# B&R Automation Studio project MotionTestBenchMaster (part 54)

```iecst
                               VAR_DOS_SEQ.Device.LTJ203.ALR_HighLimitEn := FALSE;                                     (* STEP: 89 Hema Tank Level*)
                               VAR_DOS_SEQ.Device.LTJ203.ALR_HighLimitSP := 0;
                               VAR_DOS_SEQ.Device.LTJ203.ALR_LowLimitEn := FALSE;
                               VAR_DOS_SEQ.Device.LTJ203.ALR_LowLimitSP := 0;
                               VAR_DOS_SEQ.Device.LTJ203.SP := 0;
                               VAR_DOS_SEQ.Device.LTJ203.CMP := 0;
                               VAR_DOS_SEQ.Device.LTJ203.MinDev := 0;
                               VAR_DOS_SEQ.Device.LTJ203.MaxDev := 0;

                               VAR_DOS_SEQ.Device.TTJ203.ALR_HighLimitEn := FALSE;                                     (* STEP: 89 Hema Tank Temperature*)
                               VAR_DOS_SEQ.Device.TTJ203.ALR_HighLimitSP := 0;
                               VAR_DOS_SEQ.Device.TTJ203.ALR_LowLimitEn := FALSE;
                               VAR_DOS_SEQ.Device.TTJ203.ALR_LowLimitSP := 0;
                               VAR_DOS_SEQ.Device.TTJ203.SP := 0;
                               VAR_DOS_SEQ.Device.TTJ203.CMP := 0;
                               VAR_DOS_SEQ.Device.TTJ203.MinDev := 0;
                               VAR_DOS_SEQ.Device.TTJ203.MaxDev := 0;

                               VAR_DOS_SEQ.Device.LSJ200.ALR := FALSE;                                                 (* STEP: 89 *)
                               VAR_DOS_SEQ.Device.LSJ200.WAIT_OFF := FALSE;
                               VAR_DOS_SEQ.Device.LSJ200.WAIT_ON := FALSE;

                               VAR_DOS_SEQ.Device.LSJ201.ALR := FALSE;                                                 (* STEP: 89 *)
                               VAR_DOS_SEQ.Device.LSJ201.WAIT_OFF := FALSE;
                               VAR_DOS_SEQ.Device.LSJ201.WAIT_ON := FALSE;

                               VAR_DOS_SEQ.Device.LSJ202.ALR := FALSE;                                                 (* STEP: 89 *)
                               VAR_DOS_SEQ.Device.LSJ202.WAIT_OFF := FALSE;
                               VAR_DOS_SEQ.Device.LSJ202.WAIT_ON := FALSE;

                               VAR_DOS_SEQ.Device.FSJ201.ALR := FALSE;                                                 (* STEP: 89 *)
                               VAR_DOS_SEQ.Device.FSJ201.WAIT_OFF := FALSE;
                               VAR_DOS_SEQ.Device.FSJ201.WAIT_ON := FALSE;

                               VAR_DOS_SEQ.Device.FSJ202.ALR := FALSE;                                                 (* STEP: 89 *)
                               VAR_DOS_SEQ.Device.FSJ202.WAIT_OFF := FALSE;
                               VAR_DOS_SEQ.Device.FSJ202.WAIT_ON := FALSE;

                               VAR_DOS_SEQ.Mem.PBAbortEnable := FALSE;                                                 (* STEP: 89 PB Abort Sequence Enable*)
                               VAR_DOS_SEQ.Mem.PBStopEnable := FALSE;                                                  (* STEP: 89 PB Stop Sequence Enable*)
                               VAR_DOS_SEQ.Mem.PBStartEnable := FALSE;                                                 (* STEP: 89 PB Start Sequence Enable*)
                               VAR_DOS_SEQ.Mem.ContainersStop := TRUE;                                                 (* STEP: 89 *)
                               VAR_DOS_SEQ.Mem.MachineStart := FALSE;                                                  (* STEP: 89 *)
                               VAR_DOS_SEQ.Mem.MachineStop := TRUE;                                                    (* STEP: 89 *)
                               VAR_DOS_SEQ.Mem.DummyBottles := FALSE;                                                  (* STEP: 89 Dummy Bottle Install*)
                               VAR_DOS_SEQ.Mem.PositioningRequest := TRUE;                                             (* STEP: 89 Request of Cam Positioning at height SP of Sequncer*)
                               VAR_DOS_SEQ.Mem.COP_Cycle := TRUE;                                                      (* STEP: 89 COP Cycle Check Requested*)
                               VAR_DOS_SEQ.Mem.LapsCounter := FALSE;                                                   (* STEP: 89 *)
                               VAR_DOS_SEQ.Mem.ValveOpening := FALSE;                                                  (* STEP: 89 *)
                               VAR_DOS_SEQ.Mem.CopAfterCipRequest := FALSE;                                            (* STEP: 89 Request Of Cop After Cip*)

                               VAR_DOS_SEQ.ITC.CIP_CleaningRequest := FALSE;                                           (* STEP: 89 To CIP -> Request of Solution Sending*)
                               VAR_DOS_SEQ.ITC.CIP_Alarm := FALSE;                                                     (* STEP: 89 To CIP -> Critical Alarm Present*)
                               VAR_DOS_SEQ.ITC.CIP_RinseEnded := FALSE;                                                (* STEP: 89 To CIP -> Rinse Finished*)
                               VAR_DOS_SEQ.ITC.CIP_ChangeEnded := FALSE;                                               (* STEP: 89 To CIP -> Change Finished*)
                               VAR_DOS_SEQ.ITC.CIP_DrainRunning := FALSE;                                              (* STEP: 89 To CIP -> Drain Cycle Running*)
                               VAR_DOS_SEQ.ITC.CIP_RinseRunning := FALSE;                                              (* STEP: 89 To CIP -> Rinse Cycle Running*)
                               VAR_DOS_SEQ.ITC.CIP_CleaningRunning := FALSE;                                           (* STEP: 89 To CIP -> Cleaning Cycle Running*)
                               VAR_DOS_SEQ.ITC.CIP_DrainEnded := FALSE;                                                (* STEP: 89 To CIP -> Drain Finished*)
                               VAR_DOS_SEQ.ITC.CIP_FloodingEnded := FALSE;                                             (* STEP: 89 To CIP -> Flooding Finished*)
                               VAR_DOS_SEQ.ITC.CIP_FlipEnable := FALSE;                                                (* STEP: 89 *)
                               VAR_DOS_SEQ.ITC.CIP_CycleEnded := FALSE;                                                (* STEP: 89 *)

                               VAR_DOS_SEQ.ITC.PROD_ReadyForHeating := FALSE;                                          (* STEP: 89 To PASTO -> Filler Ready for Production (Heating)*)
                               VAR_DOS_SEQ.ITC.PROD_DoserInTemperature := FALSE;                                       (* STEP: 89 To PASTO -> Filler Temperature OK (After Heating)*)
                               VAR_DOS_SEQ.ITC.PROD_ProductRequest := FALSE;                                           (* STEP: 89 To PASTO -> Product Request*)
                               VAR_DOS_SEQ.ITC.PROD_DoserOnFillingMode := FALSE;                                       (* STEP: 89 To PASTO -> Product Consumend -Filling Valve Opening*)
                               VAR_DOS_SEQ.ITC.PROD_EndProductionCompleted := FALSE;                                   (* STEP: 89 To PASTO -> End Production Done*)
                               VAR_DOS_SEQ.ITC.PROD_ProductRecoveryEnd := FALSE;                                       (* STEP: 89 To PASTO -> Product Recovery End*)
                               VAR_DOS_SEQ.ITC.PROD_WaterRequestAfterProd := FALSE;                                    (* STEP: 89 To PASTO -> Water Request For Filler Rinse Afetr Production*)

                       90: (* COP in Execution *)

                               VAR_DOS_SEQ.Device.PPJ201_PID.PID_Enable := FALSE;                                      (* STEP: 90 Doser Recovery Pump*)
                               VAR_DOS_SEQ.Device.PPJ201_PID.PID_Mode := FALSE;
                               VAR_DOS_SEQ.Device.PPJ201_PID.Auto_SP_Value := 0;
                               VAR_DOS_SEQ.Device.PPJ201_PID.FIX_Value := 0;

                               VAR_DOS_SEQ.Device.PPJ202_PID.PID_Enable := FALSE;                                      (* STEP: 90 Doser Recovery Pump*)
                               VAR_DOS_SEQ.Device.PPJ202_PID.PID_Mode := FALSE;
                               VAR_DOS_SEQ.Device.PPJ202_PID.Auto_SP_Value := 0;
                               VAR_DOS_SEQ.Device.PPJ202_PID.FIX_Value := 0;

                               VAR_DOS_SEQ.Device.PPJ203_PID.PID_Enable := FALSE;                                      (* STEP: 90 Diaphragm Pump for Recovery pulp*)
                               VAR_DOS_SEQ.Device.PPJ203_PID.PID_Mode := FALSE;
                               VAR_DOS_SEQ.Device.PPJ203_PID.Auto_SP_Value := 0;
                               VAR_DOS_SEQ.Device.PPJ203_PID.FIX_Value := 0;

                               VAR_DOS_SEQ.Device.MMJ201_PID.PID_Enable := FALSE;                                      (* STEP: 90 Shaker Motor*)
                               VAR_DOS_SEQ.Device.MMJ201_PID.PID_Mode := FALSE;
                               VAR_DOS_SEQ.Device.MMJ201_PID.Auto_SP_Value := 0;
                               VAR_DOS_SEQ.Device.MMJ201_PID.FIX_Value := 0;

                               VAR_DOS_SEQ.Device.RVJ201_PID.PID_Enable := FALSE;                                      (* STEP: 90 *)
                               VAR_DOS_SEQ.Device.RVJ201_PID.PID_Mode := FALSE;
                               VAR_DOS_SEQ.Device.RVJ201_PID.Auto_SP_Value := 0;
                               VAR_DOS_SEQ.Device.RVJ201_PID.FIX_Value := 0;

                               VAR_DOS_SEQ.Device.AVJ201.AutoCnd := FALSE;                                             (* STEP: 90 Inlet Valve*)
                               VAR_DOS_SEQ.Device.AVJ201.EnableCnd := FALSE;
                               VAR_DOS_SEQ.Device.AVJ210.AutoCnd := FALSE;                                             (* STEP: 90 Washing Duct Valve*)
                               VAR_DOS_SEQ.Device.AVJ210.EnableCnd := FALSE;
                               VAR_DOS_SEQ.Device.AVJ211.AutoCnd := FALSE;                                             (* STEP: 90 Sprayball Valve*)
                               VAR_DOS_SEQ.Device.AVJ211.EnableCnd := FALSE;
                               VAR_DOS_SEQ.Device.AVJ212.AutoCnd := FALSE;                                             (* STEP: 90 *)
                               VAR_DOS_SEQ.Device.AVJ212.EnableCnd := FALSE;
                               VAR_DOS_SEQ.Device.AVJ215.AutoCnd := TRUE;                                              (* STEP: 90 Atmospheric drain valve*)
                               VAR_DOS_SEQ.Device.AVJ215.EnableCnd := FALSE;
                               VAR_DOS_SEQ.Device.AVJ216.AutoCnd := FALSE;                                             (* STEP: 90 Recirculation Valve*)
                               VAR_DOS_SEQ.Device.AVJ216.EnableCnd := FALSE;
                               VAR_DOS_SEQ.Device.AVJ217.AutoCnd := TRUE;                                              (* STEP: 90 Tank Hema Drain Valve*)
                               VAR_DOS_SEQ.Device.AVJ217.EnableCnd := FALSE;
                               VAR_DOS_SEQ.Device.AVJ218.AutoCnd := FALSE;                                             (* STEP: 90 Recirculation Valve*)
                               VAR_DOS_SEQ.Device.AVJ218.EnableCnd := FALSE;
                               VAR_DOS_SEQ.Device.AVJ221.AutoCnd := FALSE;                                             (* STEP: 90 Inlet Loop Valve*)
                               VAR_DOS_SEQ.Device.AVJ221.EnableCnd := FALSE;
                               VAR_DOS_SEQ.Device.AVJ230.AutoCnd := FALSE;                                             (* STEP: 90 *)
                               VAR_DOS_SEQ.Device.AVJ230.EnableCnd := FALSE;
                               VAR_DOS_SEQ.Device.AVJ231.AutoCnd := FALSE;                                             (* STEP: 90 *)
                               VAR_DOS_SEQ.Device.AVJ231.EnableCnd := FALSE;
                               VAR_DOS_SEQ.Device.AVJ232.AutoCnd := FALSE;                                             (* STEP: 90 *)
                               VAR_DOS_SEQ.Device.AVJ232.EnableCnd := FALSE;
                               VAR_DOS_SEQ.Device.AVJ233.AutoCnd := FALSE;                                             (* STEP: 90 *)
                               VAR_DOS_SEQ.Device.AVJ233.EnableCnd := FALSE;
                               VAR_DOS_SEQ.Device.AVJ234.AutoCnd := FALSE;                                             (* STEP: 90 *)
                               VAR_DOS_SEQ.Device.AVJ234.EnableCnd := FALSE;
                               VAR_DOS_SEQ.Device.AVJ235.AutoCnd := FALSE;                                             (* STEP: 90 *)
                               VAR_DOS_SEQ.Device.AVJ235.EnableCnd := FALSE;

                               VAR_DOS_SEQ.Device.LTJ203.ALR_HighLimitEn := FALSE;                                     (* STEP: 90 Hema Tank Level*)
                               VAR_DOS_SEQ.Device.LTJ203.ALR_HighLimitSP := 0;
                               VAR_DOS_SEQ.Device.LTJ203.ALR_LowLimitEn := FALSE;
                               VAR_DOS_SEQ.Device.LTJ203.ALR_LowLimitSP := 0;
                               VAR_DOS_SEQ.Device.LTJ203.SP := 0;
                               VAR_DOS_SEQ.Device.LTJ203.CMP := 0;
                               VAR_DOS_SEQ.Device.LTJ203.MinDev := 0;
                               VAR_DOS_SEQ.Device.LTJ203.MaxDev := 0;

                               VAR_DOS_SEQ.Device.TTJ203.ALR_HighLimitEn := FALSE;                                     (* STEP: 90 Hema Tank Temperature*)
                               VAR_DOS_SEQ.Device.TTJ203.ALR_HighLimitSP := 0;
                               VAR_DOS_SEQ.Device.TTJ203.ALR_LowLimitEn := FALSE;
                               VAR_DOS_SEQ.Device.TTJ203.ALR_LowLimitSP := 0;
                               VAR_DOS_SEQ.Device.TTJ203.SP := 0;
                               VAR_DOS_SEQ.Device.TTJ203.CMP := 0;
                               VAR_DOS_SEQ.Device.TTJ203.MinDev := 0;
                               VAR_DOS_SEQ.Device.TTJ203.MaxDev := 0;

                               VAR_DOS_SEQ.Device.LSJ200.ALR := FALSE;                                                 (* STEP: 90 *)
                               VAR_DOS_SEQ.Device.LSJ200.WAIT_OFF := FALSE;
                               VAR_DOS_SEQ.Device.LSJ200.WAIT_ON := FALSE;

                               VAR_DOS_SEQ.Device.LSJ201.ALR := FALSE;                                                 (* STEP: 90 *)
                               VAR_DOS_SEQ.Device.LSJ201.WAIT_OFF := FALSE;
                               VAR_DOS_SEQ.Device.LSJ201.WAIT_ON := FALSE;

                               VAR_DOS_SEQ.Device.LSJ202.ALR := FALSE;                                                 (* STEP: 90 *)
                               VAR_DOS_SEQ.Device.LSJ202.WAIT_OFF := FALSE;
                               VAR_DOS_SEQ.Device.LSJ202.WAIT_ON := FALSE;

                               VAR_DOS_SEQ.Device.FSJ201.ALR := FALSE;                                                 (* STEP: 90 *)
                               VAR_DOS_SEQ.Device.FSJ201.WAIT_OFF := FALSE;
                               VAR_DOS_SEQ.Device.FSJ201.WAIT_ON := FALSE;

                               VAR_DOS_SEQ.Device.FSJ202.ALR := FALSE;                                                 (* STEP: 90 *)
                               VAR_DOS_SEQ.Device.FSJ202.WAIT_OFF := FALSE;
                               VAR_DOS_SEQ.Device.FSJ202.WAIT_ON := FALSE;

                               VAR_DOS_SEQ.Mem.PBAbortEnable := FALSE;                                                 (* STEP: 90 PB Abort Sequence Enable*)
                               VAR_DOS_SEQ.Mem.PBStopEnable := FALSE;                                                  (* STEP: 90 PB Stop Sequence Enable*)
                               VAR_DOS_SEQ.Mem.PBStartEnable := FALSE;                                                 (* STEP: 90 PB Start Sequence Enable*)
                               VAR_DOS_SEQ.Mem.ContainersStop := TRUE;                                                 (* STEP: 90 *)
                               VAR_DOS_SEQ.Mem.MachineStart := TRUE;                                                   (* STEP: 90 *)
                               VAR_DOS_SEQ.Mem.MachineStop := FALSE;                                                   (* STEP: 90 *)
                               VAR_DOS_SEQ.Mem.DummyBottles := FALSE;                                                  (* STEP: 90 Dummy Bottle Install*)
                               VAR_DOS_SEQ.Mem.PositioningRequest := FALSE;                                            (* STEP: 90 Request of Cam Positioning at height SP of Sequncer*)
                               VAR_DOS_SEQ.Mem.COP_Cycle := TRUE;                                                      (* STEP: 90 COP Cycle Check Requested*)
                               VAR_DOS_SEQ.Mem.LapsCounter := FALSE;                                                   (* STEP: 90 *)
                               VAR_DOS_SEQ.Mem.ValveOpening := FALSE;                                                  (* STEP: 90 *)
                               VAR_DOS_SEQ.Mem.CopAfterCipRequest := FALSE;                                            (* STEP: 90 Request Of Cop After Cip*)

                               VAR_DOS_SEQ.ITC.CIP_CleaningRequest := FALSE;                                           (* STEP: 90 To CIP -> Request of Solution Sending*)
                               VAR_DOS_SEQ.ITC.CIP_Alarm := FALSE;                                                     (* STEP: 90 To CIP -> Critical Alarm Present*)
                               VAR_DOS_SEQ.ITC.CIP_RinseEnded := FALSE;                                                (* STEP: 90 To CIP -> Rinse Finished*)
                               VAR_DOS_SEQ.ITC.CIP_ChangeEnded := FALSE;                                               (* STEP: 90 To CIP -> Change Finished*)
                               VAR_DOS_SEQ.ITC.CIP_DrainRunning := FALSE;                                              (* STEP: 90 To CIP -> Drain Cycle Running*)
                               VAR_DOS_SEQ.ITC.CIP_RinseRunning := FALSE;                                              (* STEP: 90 To CIP -> Rinse Cycle Running*)
                               VAR_DOS_SEQ.ITC.CIP_CleaningRunning := FALSE;                                           (* STEP: 90 To CIP -> Cleaning Cycle Running*)
                               VAR_DOS_SEQ.ITC.CIP_DrainEnded := FALSE;                                                (* STEP: 90 To CIP -> Drain Finished*)
                               VAR_DOS_SEQ.ITC.CIP_FloodingEnded := FALSE;                                             (* STEP: 90 To CIP -> Flooding Finished*)
                               VAR_DOS_SEQ.ITC.CIP_FlipEnable := FALSE;                                                (* STEP: 90 *)
                               VAR_DOS_SEQ.ITC.CIP_CycleEnded := FALSE;                                                (* STEP: 90 *)

                               VAR_DOS_SEQ.ITC.PROD_ReadyForHeating := FALSE;                                          (* STEP: 90 To PASTO -> Filler Ready for Production (Heating)*)
                               VAR_DOS_SEQ.ITC.PROD_DoserInTemperature := FALSE;                                       (* STEP: 90 To PASTO -> Filler Temperature OK (After Heating)*)
                               VAR_DOS_SEQ.ITC.PROD_ProductRequest := FALSE;                                           (* STEP: 90 To PASTO -> Product Request*)
                               VAR_DOS_SEQ.ITC.PROD_DoserOnFillingMode := FALSE;                                       (* STEP: 90 To PASTO -> Product Consumend -Filling Valve Opening*)
                               VAR_DOS_SEQ.ITC.PROD_EndProductionCompleted := FALSE;                                   (* STEP: 90 To PASTO -> End Production Done*)
                               VAR_DOS_SEQ.ITC.PROD_ProductRecoveryEnd := FALSE;                                       (* STEP: 90 To PASTO -> Product Recovery End*)
                               VAR_DOS_SEQ.ITC.PROD_WaterRequestAfterProd := FALSE;                                    (* STEP: 90 To PASTO -> Water Request For Filler Rinse Afetr Production*)
//change
                       91: (* Drain Recovery Skid *)

								VAR_DOS_SEQ.Device.PPJ201_PID.PID_Enable := FALSE;                                      (* STEP: 91 Doser Recovery Pump*)
								VAR_DOS_SEQ.Device.PPJ201_PID.PID_Mode := FALSE;
								VAR_DOS_SEQ.Device.PPJ201_PID.Auto_SP_Value := 0;
								VAR_DOS_SEQ.Device.PPJ201_PID.FIX_Value := 0;

								VAR_DOS_SEQ.Device.PPJ202_PID.PID_Enable := FALSE;                                      (* STEP: 91 Doser Recovery Pump*)
								VAR_DOS_SEQ.Device.PPJ202_PID.PID_Mode := FALSE;
								VAR_DOS_SEQ.Device.PPJ202_PID.Auto_SP_Value := 0;
								VAR_DOS_SEQ.Device.PPJ202_PID.FIX_Value := 0;

								VAR_DOS_SEQ.Device.PPJ203_PID.PID_Enable := FALSE;                                      (* STEP: 91 Diaphragm Pump for Recovery pulp*)
								VAR_DOS_SEQ.Device.PPJ203_PID.PID_Mode := FALSE;
								VAR_DOS_SEQ.Device.PPJ203_PID.Auto_SP_Value := 0;
								VAR_DOS_SEQ.Device.PPJ203_PID.FIX_Value := 0;

								VAR_DOS_SEQ.Device.MMJ201_PID.PID_Enable := FALSE;                                      (* STEP: 91 Shaker Motor*)
								VAR_DOS_SEQ.Device.MMJ201_PID.PID_Mode := FALSE;
								VAR_DOS_SEQ.Device.MMJ201_PID.Auto_SP_Value := 0;
								VAR_DOS_SEQ.Device.MMJ201_PID.FIX_Value := 0;

								VAR_DOS_SEQ.Device.RVJ201_PID.PID_Enable := FALSE;                                      (* STEP: 91 *)
								VAR_DOS_SEQ.Device.RVJ201_PID.PID_Mode := FALSE;
								VAR_DOS_SEQ.Device.RVJ201_PID.Auto_SP_Value := 0;
								VAR_DOS_SEQ.Device.RVJ201_PID.FIX_Value := 0;

								VAR_DOS_SEQ.Device.AVJ201.AutoCnd := FALSE;                                             (* STEP: 91 Inlet Valve*)
								VAR_DOS_SEQ.Device.AVJ201.EnableCnd := FALSE;
								VAR_DOS_SEQ.Device.AVJ210.AutoCnd := FALSE;                                             (* STEP: 91 Washing Duct Valve*)
								VAR_DOS_SEQ.Device.AVJ210.EnableCnd := FALSE;
								VAR_DOS_SEQ.Device.AVJ211.AutoCnd := FALSE;                                             (* STEP: 91 Sprayball Valve*)
								VAR_DOS_SEQ.Device.AVJ211.EnableCnd := FALSE;
								VAR_DOS_SEQ.Device.AVJ212.AutoCnd := FALSE;                                             (* STEP: 91 *)
								VAR_DOS_SEQ.Device.AVJ212.EnableCnd := FALSE;
								VAR_DOS_SEQ.Device.AVJ215.AutoCnd := TRUE;                                              (* STEP: 91 Atmospheric drain valve*)
								VAR_DOS_SEQ.Device.AVJ215.EnableCnd := FALSE;
								VAR_DOS_SEQ.Device.AVJ216.AutoCnd := FALSE;                                             (* STEP: 91 Recirculation Valve*)
								VAR_DOS_SEQ.Device.AVJ216.EnableCnd := FALSE;
								VAR_DOS_SEQ.Device.AVJ217.AutoCnd := TRUE;                                              (* STEP: 91 Tank Hema Drain Valve*)
								VAR_DOS_SEQ.Device.AVJ217.EnableCnd := FALSE;
								VAR_DOS_SEQ.Device.AVJ218.AutoCnd := FALSE;                                             (* STEP: 91 Recirculation Valve*)
								VAR_DOS_SEQ.Device.AVJ218.EnableCnd := FALSE;
								VAR_DOS_SEQ.Device.AVJ221.AutoCnd := FALSE;                                             (* STEP: 91 Inlet Loop Valve*)
								VAR_DOS_SEQ.Device.AVJ221.EnableCnd := FALSE;
								VAR_DOS_SEQ.Device.AVJ230.AutoCnd := FALSE;                                             (* STEP: 91 *)
								VAR_DOS_SEQ.Device.AVJ230.EnableCnd := FALSE;
								VAR_DOS_SEQ.Device.AVJ231.AutoCnd := FALSE;                                             (* STEP: 91 *)
								VAR_DOS_SEQ.Device.AVJ231.EnableCnd := FALSE;
								VAR_DOS_SEQ.Device.AVJ232.AutoCnd := TRUE;                                             (* STEP: 91 *)
								VAR_DOS_SEQ.Device.AVJ232.EnableCnd := FALSE;
								VAR_DOS_SEQ.Device.AVJ233.AutoCnd := FALSE;                                             (* STEP: 91 *)
								VAR_DOS_SEQ.Device.AVJ233.EnableCnd := FALSE;
								VAR_DOS_SEQ.Device.AVJ234.AutoCnd := FALSE;                                             (* STEP: 91 *)
								VAR_DOS_SEQ.Device.AVJ234.EnableCnd := FALSE;
								VAR_DOS_SEQ.Device.AVJ235.AutoCnd := TRUE;                                             (* STEP: 91 *)
								VAR_DOS_SEQ.Device.AVJ235.EnableCnd := FALSE;

								VAR_DOS_SEQ.Device.LTJ203.ALR_HighLimitEn := FALSE;                                     (* STEP: 91 Hema Tank Level*)
								VAR_DOS_SEQ.Device.LTJ203.ALR_HighLimitSP := 0;
								VAR_DOS_SEQ.Device.LTJ203.ALR_LowLimitEn := FALSE;
								VAR_DOS_SEQ.Device.LTJ203.ALR_LowLimitSP := 0;
								VAR_DOS_SEQ.Device.LTJ203.SP := 0;
								VAR_DOS_SEQ.Device.LTJ203.CMP := 0;
								VAR_DOS_SEQ.Device.LTJ203.MinDev := 0;
								VAR_DOS_SEQ.Device.LTJ203.MaxDev := 0;

								VAR_DOS_SEQ.Device.TTJ203.ALR_HighLimitEn := FALSE;                                     (* STEP: 91 Hema Tank Temperature*)
								VAR_DOS_SEQ.Device.TTJ203.ALR_HighLimitSP := 0;
								VAR_DOS_SEQ.Device.TTJ203.ALR_LowLimitEn := FALSE;
								VAR_DOS_SEQ.Device.TTJ203.ALR_LowLimitSP := 0;
								VAR_DOS_SEQ.Device.TTJ203.SP := 0;
								VAR_DOS_SEQ.Device.TTJ203.CMP := 0;
								VAR_DOS_SEQ.Device.TTJ203.MinDev := 0;
								VAR_DOS_SEQ.Device.TTJ203.MaxDev := 0;

								VAR_DOS_SEQ.Device.LSJ200.ALR := FALSE;                                                 (* STEP: 91 *)
								VAR_DOS_SEQ.Device.LSJ200.WAIT_OFF := FALSE;
								VAR_DOS_SEQ.Device.LSJ200.WAIT_ON := FALSE;

								VAR_DOS_SEQ.Device.LSJ201.ALR := FALSE;                                                 (* STEP: 91 *)
								VAR_DOS_SEQ.Device.LSJ201.WAIT_OFF := FALSE;
								VAR_DOS_SEQ.Device.LSJ201.WAIT_ON := FALSE;

								VAR_DOS_SEQ.Device.LSJ202.ALR := FALSE;                                                 (* STEP: 91 *)
								VAR_DOS_SEQ.Device.LSJ202.WAIT_OFF := FALSE;
								VAR_DOS_SEQ.Device.LSJ202.WAIT_ON := FALSE;

								VAR_DOS_SEQ.Device.FSJ201.ALR := FALSE;                                                 (* STEP: 91 *)
								VAR_DOS_SEQ.Device.FSJ201.WAIT_OFF := FALSE;
								VAR_DOS_SEQ.Device.FSJ201.WAIT_ON := FALSE;

								VAR_DOS_SEQ.Device.FSJ202.ALR := FALSE;                                                 (* STEP: 91 *)
								VAR_DOS_SEQ.Device.FSJ202.WAIT_OFF := FALSE;
								VAR_DOS_SEQ.Device.FSJ202.WAIT_ON := FALSE;

								VAR_DOS_SEQ.Mem.PBAbortEnable := FALSE;                                                 (* STEP: 91 PB Abort Sequence Enable*)
								VAR_DOS_SEQ.Mem.PBStopEnable := FALSE;                                                  (* STEP: 91 PB Stop Sequence Enable*)
								VAR_DOS_SEQ.Mem.PBStartEnable := FALSE;                                                 (* STEP: 91 PB Start Sequence Enable*)
								VAR_DOS_SEQ.Mem.ContainersStop := TRUE;                                                 (* STEP: 91 *)
								VAR_DOS_SEQ.Mem.MachineStart := FALSE;                                                   (* STEP: 91 *)
								VAR_DOS_SEQ.Mem.MachineStop := TRUE;                                                   (* STEP: 91 *)
								VAR_DOS_SEQ.Mem.DummyBottles := FALSE;                                                  (* STEP: 91 Dummy Bottle Install*)
								VAR_DOS_SEQ.Mem.PositioningRequest := FALSE;                                            (* STEP: 91 Request of Cam Positioning at height SP of Sequncer*)
								VAR_DOS_SEQ.Mem.COP_Cycle := TRUE;                                                      (* STEP: 91 COP Cycle Check Requested*)
								VAR_DOS_SEQ.Mem.LapsCounter := FALSE;                                                   (* STEP: 91 *)
								VAR_DOS_SEQ.Mem.ValveOpening := FALSE;                                                  (* STEP: 91 *)
								VAR_DOS_SEQ.Mem.CopAfterCipRequest := FALSE;                                            (* STEP: 91 Request Of Cop After Cip*)

								VAR_DOS_SEQ.ITC.CIP_CleaningRequest := FALSE;                                           (* STEP: 91 To CIP -> Request of Solution Sending*)
								VAR_DOS_SEQ.ITC.CIP_Alarm := FALSE;                                                     (* STEP: 91 To CIP -> Critical Alarm Present*)
								VAR_DOS_SEQ.ITC.CIP_RinseEnded := FALSE;                                                (* STEP: 91 To CIP -> Rinse Finished*)
								VAR_DOS_SEQ.ITC.CIP_ChangeEnded := FALSE;                                               (* STEP: 91 To CIP -> Change Finished*)
								VAR_DOS_SEQ.ITC.CIP_DrainRunning := FALSE;                                              (* STEP: 91 To CIP -> Drain Cycle Running*)
								VAR_DOS_SEQ.ITC.CIP_RinseRunning := FALSE;                                              (* STEP: 91 To CIP -> Rinse Cycle Running*)
								VAR_DOS_SEQ.ITC.CIP_CleaningRunning := FALSE;                                           (* STEP: 91 To CIP -> Cleaning Cycle Running*)
								VAR_DOS_SEQ.ITC.CIP_DrainEnded := FALSE;                                                (* STEP: 91 To CIP -> Drain Finished*)
								VAR_DOS_SEQ.ITC.CIP_FloodingEnded := FALSE;                                             (* STEP: 91 To CIP -> Flooding Finished*)
								VAR_DOS_SEQ.ITC.CIP_FlipEnable := FALSE;                                                (* STEP: 91 *)
								VAR_DOS_SEQ.ITC.CIP_CycleEnded := FALSE;                                                (* STEP: 91 *)

								VAR_DOS_SEQ.ITC.PROD_ReadyForHeating := FALSE;                                          (* STEP: 91 To PASTO -> Filler Ready for Production (Heating)*)
								VAR_DOS_SEQ.ITC.PROD_DoserInTemperature := FALSE;                                       (* STEP: 91 To PASTO -> Filler Temperature OK (After Heating)*)
								VAR_DOS_SEQ.ITC.PROD_ProductRequest := FALSE;                                           (* STEP: 91 To PASTO -> Product Request*)
								VAR_DOS_SEQ.ITC.PROD_DoserOnFillingMode := FALSE;                                       (* STEP: 91 To PASTO -> Product Consumend -Filling Valve Opening*)
								VAR_DOS_SEQ.ITC.PROD_EndProductionCompleted := FALSE;                                   (* STEP: 91 To PASTO -> End Production Done*)
								VAR_DOS_SEQ.ITC.PROD_ProductRecoveryEnd := FALSE;                                       (* STEP: 91 To PASTO -> Product Recovery End*)
								VAR_DOS_SEQ.ITC.PROD_WaterRequestAfterProd := FALSE;                                    (* STEP: 91 To PASTO -> Water Request For Filler Rinse Afetr Production*)

                       92: (* CIP -Wait Dummy Bottles Disinsertion *)

                               VAR_DOS_SEQ.Device.PPJ201_PID.PID_Enable := FALSE;                                      (* STEP: 92 Doser Recovery Pump*)
                               VAR_DOS_SEQ.Device.PPJ201_PID.PID_Mode := FALSE;
                               VAR_DOS_SEQ.Device.PPJ201_PID.Auto_SP_Value := 0;
                               VAR_DOS_SEQ.Device.PPJ201_PID.FIX_Value := 0;

                               VAR_DOS_SEQ.Device.PPJ202_PID.PID_Enable := FALSE;                                      (* STEP: 92 Doser Recovery Pump*)
                               VAR_DOS_SEQ.Device.PPJ202_PID.PID_Mode := FALSE;
                               VAR_DOS_SEQ.Device.PPJ202_PID.Auto_SP_Value := 0;
                               VAR_DOS_SEQ.Device.PPJ202_PID.FIX_Value := 0;

                               VAR_DOS_SEQ.Device.PPJ203_PID.PID_Enable := FALSE;                                      (* STEP: 92 Diaphragm Pump for Recovery pulp*)
                               VAR_DOS_SEQ.Device.PPJ203_PID.PID_Mode := FALSE;
                               VAR_DOS_SEQ.Device.PPJ203_PID.Auto_SP_Value := 0;
                               VAR_DOS_SEQ.Device.PPJ203_PID.FIX_Value := 0;

                               VAR_DOS_SEQ.Device.MMJ201_PID.PID_Enable := FALSE;                                      (* STEP: 92 Shaker Motor*)
                               VAR_DOS_SEQ.Device.MMJ201_PID.PID_Mode := FALSE;
                               VAR_DOS_SEQ.Device.MMJ201_PID.Auto_SP_Value := 0;
                               VAR_DOS_SEQ.Device.MMJ201_PID.FIX_Value := 0;

                               VAR_DOS_SEQ.Device.RVJ201_PID.PID_Enable := FALSE;                                      (* STEP: 92 *)
                               VAR_DOS_SEQ.Device.RVJ201_PID.PID_Mode := FALSE;
                               VAR_DOS_SEQ.Device.RVJ201_PID.Auto_SP_Value := 0;
                               VAR_DOS_SEQ.Device.RVJ201_PID.FIX_Value := 0;

                               VAR_DOS_SEQ.Device.AVJ201.AutoCnd := FALSE;                                             (* STEP: 92 Inlet Valve*)
                               VAR_DOS_SEQ.Device.AVJ201.EnableCnd := FALSE;
                               VAR_DOS_SEQ.Device.AVJ210.AutoCnd := FALSE;                                             (* STEP: 92 Washing Duct Valve*)
                               VAR_DOS_SEQ.Device.AVJ210.EnableCnd := FALSE;
                               VAR_DOS_SEQ.Device.AVJ211.AutoCnd := FALSE;                                             (* STEP: 92 Sprayball Valve*)
                               VAR_DOS_SEQ.Device.AVJ211.EnableCnd := FALSE;
                               VAR_DOS_SEQ.Device.AVJ212.AutoCnd := FALSE;                                             (* STEP: 92 *)
                               VAR_DOS_SEQ.Device.AVJ212.EnableCnd := FALSE;
                               VAR_DOS_SEQ.Device.AVJ215.AutoCnd := FALSE;                                             (* STEP: 92 Atmospheric drain valve*)
                               VAR_DOS_SEQ.Device.AVJ215.EnableCnd := FALSE;
                               VAR_DOS_SEQ.Device.AVJ216.AutoCnd := FALSE;                                             (* STEP: 92 Recirculation Valve*)
                               VAR_DOS_SEQ.Device.AVJ216.EnableCnd := FALSE;
                               VAR_DOS_SEQ.Device.AVJ217.AutoCnd := FALSE;                                             (* STEP: 92 Tank Hema Drain Valve*)
                               VAR_DOS_SEQ.Device.AVJ217.EnableCnd := FALSE;
                               VAR_DOS_SEQ.Device.AVJ218.AutoCnd := FALSE;                                             (* STEP: 92 Recirculation Valve*)
                               VAR_DOS_SEQ.Device.AVJ218.EnableCnd := FALSE;
                               VAR_DOS_SEQ.Device.AVJ221.AutoCnd := FALSE;                                             (* STEP: 92 Inlet Loop Valve*)
                               VAR_DOS_SEQ.Device.AVJ221.EnableCnd := FALSE;
                               VAR_DOS_SEQ.Device.AVJ230.AutoCnd := FALSE;                                             (* STEP: 92 *)
                               VAR_DOS_SEQ.Device.AVJ230.EnableCnd := FALSE;
                               VAR_DOS_SEQ.Device.AVJ231.AutoCnd := FALSE;                                             (* STEP: 92 *)
                               VAR_DOS_SEQ.Device.AVJ231.EnableCnd := FALSE;
                               VAR_DOS_SEQ.Device.AVJ232.AutoCnd := FALSE;                                             (* STEP: 92 *)
                               VAR_DOS_SEQ.Device.AVJ232.EnableCnd := FALSE;
                               VAR_DOS_SEQ.Device.AVJ233.AutoCnd := FALSE;                                             (* STEP: 92 *)
                               VAR_DOS_SEQ.Device.AVJ233.EnableCnd := FALSE;
                               VAR_DOS_SEQ.Device.AVJ234.AutoCnd := FALSE;                                             (* STEP: 92 *)
                               VAR_DOS_SEQ.Device.AVJ234.EnableCnd := FALSE;
                               VAR_DOS_SEQ.Device.AVJ235.AutoCnd := FALSE;                                             (* STEP: 92 *)
                               VAR_DOS_SEQ.Device.AVJ235.EnableCnd := FALSE;

                               VAR_DOS_SEQ.Device.LTJ203.ALR_HighLimitEn := FALSE;                                     (* STEP: 92 Hema Tank Level*)
                               VAR_DOS_SEQ.Device.LTJ203.ALR_HighLimitSP := 0;
                               VAR_DOS_SEQ.Device.LTJ203.ALR_LowLimitEn := FALSE;
                               VAR_DOS_SEQ.Device.LTJ203.ALR_LowLimitSP := 0;
                               VAR_DOS_SEQ.Device.LTJ203.SP := 0;
                               VAR_DOS_SEQ.Device.LTJ203.CMP := 0;
                               VAR_DOS_SEQ.Device.LTJ203.MinDev := 0;
                               VAR_DOS_SEQ.Device.LTJ203.MaxDev := 0;

                               VAR_DOS_SEQ.Device.TTJ203.ALR_HighLimitEn := FALSE;                                     (* STEP: 92 Hema Tank Temperature*)
                               VAR_DOS_SEQ.Device.TTJ203.ALR_HighLimitSP := 0;
                               VAR_DOS_SEQ.Device.TTJ203.ALR_LowLimitEn := FALSE;
                               VAR_DOS_SEQ.Device.TTJ203.ALR_LowLimitSP := 0;
                               VAR_DOS_SEQ.Device.TTJ203.SP := 0;
                               VAR_DOS_SEQ.Device.TTJ203.CMP := 0;
                               VAR_DOS_SEQ.Device.TTJ203.MinDev := 0;
                               VAR_DOS_SEQ.Device.TTJ203.MaxDev := 0;

                               VAR_DOS_SEQ.Device.LSJ200.ALR := FALSE;                                                 (* STEP: 92 *)
                               VAR_DOS_SEQ.Device.LSJ200.WAIT_OFF := FALSE;
                               VAR_DOS_SEQ.Device.LSJ200.WAIT_ON := FALSE;

                               VAR_DOS_SEQ.Device.LSJ201.ALR := FALSE;                                                 (* STEP: 92 *)
                               VAR_DOS_SEQ.Device.LSJ201.WAIT_OFF := FALSE;
                               VAR_DOS_SEQ.Device.LSJ201.WAIT_ON := FALSE;

                               VAR_DOS_SEQ.Device.LSJ202.ALR := FALSE;                                                 (* STEP: 92 *)
                               VAR_DOS_SEQ.Device.LSJ202.WAIT_OFF := FALSE;
                               VAR_DOS_SEQ.Device.LSJ202.WAIT_ON := FALSE;

                               VAR_DOS_SEQ.Device.FSJ201.ALR := FALSE;                                                 (* STEP: 92 *)
                               VAR_DOS_SEQ.Device.FSJ201.WAIT_OFF := FALSE;
                               VAR_DOS_SEQ.Device.FSJ201.WAIT_ON := FALSE;

                               VAR_DOS_SEQ.Device.FSJ202.ALR := FALSE;                                                 (* STEP: 92 *)
                               VAR_DOS_SEQ.Device.FSJ202.WAIT_OFF := FALSE;
                               VAR_DOS_SEQ.Device.FSJ202.WAIT_ON := FALSE;

                               VAR_DOS_SEQ.Mem.PBAbortEnable := FALSE;                                                 (* STEP: 92 PB Abort Sequence Enable*)
                               VAR_DOS_SEQ.Mem.PBStopEnable := FALSE;                                                  (* STEP: 92 PB Stop Sequence Enable*)
                               VAR_DOS_SEQ.Mem.PBStartEnable := FALSE;                                                 (* STEP: 92 PB Start Sequence Enable*)
                               VAR_DOS_SEQ.Mem.ContainersStop := FALSE;                                                (* STEP: 92 *)
                               VAR_DOS_SEQ.Mem.MachineStart := FALSE;                                                  (* STEP: 92 *)
                               VAR_DOS_SEQ.Mem.MachineStop := FALSE;                                                   (* STEP: 92 *)
                               VAR_DOS_SEQ.Mem.DummyBottles := FALSE;                                                  (* STEP: 92 Dummy Bottle Install*)
                               VAR_DOS_SEQ.Mem.PositioningRequest := FALSE;                                            (* STEP: 92 Request of Cam Positioning at height SP of Sequncer*)
                               VAR_DOS_SEQ.Mem.COP_Cycle := FALSE;                                                     (* STEP: 92 COP Cycle Check Requested*)
                               VAR_DOS_SEQ.Mem.LapsCounter := FALSE;                                                   (* STEP: 92 *)
                               VAR_DOS_SEQ.Mem.ValveOpening := FALSE;                                                  (* STEP: 92 *)
                               VAR_DOS_SEQ.Mem.CopAfterCipRequest := FALSE;                                            (* STEP: 92 Request Of Cop After Cip*)

                               VAR_DOS_SEQ.ITC.CIP_CleaningRequest := FALSE;                                           (* STEP: 92 To CIP -> Request of Solution Sending*)
                               VAR_DOS_SEQ.ITC.CIP_Alarm := FALSE;                                                     (* STEP: 92 To CIP -> Critical Alarm Present*)
                               VAR_DOS_SEQ.ITC.CIP_RinseEnded := FALSE;                                                (* STEP: 92 To CIP -> Rinse Finished*)
                               VAR_DOS_SEQ.ITC.CIP_ChangeEnded := FALSE;                                               (* STEP: 92 To CIP -> Change Finished*)
                               VAR_DOS_SEQ.ITC.CIP_DrainRunning := FALSE;                                              (* STEP: 92 To CIP -> Drain Cycle Running*)
                               VAR_DOS_SEQ.ITC.CIP_RinseRunning := FALSE;                                              (* STEP: 92 To CIP -> Rinse Cycle Running*)
                               VAR_DOS_SEQ.ITC.CIP_CleaningRunning := FALSE;                                           (* STEP: 92 To CIP -> Cleaning Cycle Running*)
                               VAR_DOS_SEQ.ITC.CIP_DrainEnded := FALSE;                                                (* STEP: 92 To CIP -> Drain Finished*)
                               VAR_DOS_SEQ.ITC.CIP_FloodingEnded := FALSE;                                             (* STEP: 92 To CIP -> Flooding Finished*)
                               VAR_DOS_SEQ.ITC.CIP_FlipEnable := FALSE;                                                (* STEP: 92 *)
                               VAR_DOS_SEQ.ITC.CIP_CycleEnded := FALSE;                                                (* STEP: 92 *)

                               VAR_DOS_SEQ.ITC.PROD_ReadyForHeating := FALSE;                                          (* STEP: 92 To PASTO -> Filler Ready for Production (Heating)*)
                               VAR_DOS_SEQ.ITC.PROD_DoserInTemperature := FALSE;                                       (* STEP: 92 To PASTO -> Filler Temperature OK (After Heating)*)
                               VAR_DOS_SEQ.ITC.PROD_ProductRequest := FALSE;                                           (* STEP: 92 To PASTO -> Product Request*)
                               VAR_DOS_SEQ.ITC.PROD_DoserOnFillingMode := FALSE;                                       (* STEP: 92 To PASTO -> Product Consumend -Filling Valve Opening*)
                               VAR_DOS_SEQ.ITC.PROD_EndProductionCompleted := FALSE;                                   (* STEP: 92 To PASTO -> End Production Done*)
                               VAR_DOS_SEQ.ITC.PROD_ProductRecoveryEnd := FALSE;                                       (* STEP: 92 To PASTO -> Product Recovery End*)
                               VAR_DOS_SEQ.ITC.PROD_WaterRequestAfterProd := FALSE;                                    (* STEP: 92 To PASTO -> Water Request For Filler Rinse Afetr Production*)

                       93..94: (* Spare Steps *)

                       95: (* CIP - Stopped *)

                               VAR_DOS_SEQ.Device.PPJ201_PID.PID_Enable := FALSE;                                      (* STEP: 95 Doser Recovery Pump*)
                               VAR_DOS_SEQ.Device.PPJ201_PID.PID_Mode := FALSE;
                               VAR_DOS_SEQ.Device.PPJ201_PID.Auto_SP_Value := 0;
                               VAR_DOS_SEQ.Device.PPJ201_PID.FIX_Value := 0;

                               VAR_DOS_SEQ.Device.PPJ202_PID.PID_Enable := FALSE;                                      (* STEP: 95 Doser Recovery Pump*)
                               VAR_DOS_SEQ.Device.PPJ202_PID.PID_Mode := FALSE;
                               VAR_DOS_SEQ.Device.PPJ202_PID.Auto_SP_Value := 0;
                               VAR_DOS_SEQ.Device.PPJ202_PID.FIX_Value := 0;

                               VAR_DOS_SEQ.Device.PPJ203_PID.PID_Enable := FALSE;                                      (* STEP: 95 Diaphragm Pump for Recovery pulp*)
                               VAR_DOS_SEQ.Device.PPJ203_PID.PID_Mode := FALSE;
                               VAR_DOS_SEQ.Device.PPJ203_PID.Auto_SP_Value := 0;
                               VAR_DOS_SEQ.Device.PPJ203_PID.FIX_Value := 0;

                               VAR_DOS_SEQ.Device.MMJ201_PID.PID_Enable := FALSE;                                      (* STEP: 95 Shaker Motor*)
                               VAR_DOS_SEQ.Device.MMJ201_PID.PID_Mode := FALSE;
                               VAR_DOS_SEQ.Device.MMJ201_PID.Auto_SP_Value := 0;
                               VAR_DOS_SEQ.Device.MMJ201_PID.FIX_Value := 0;

                               VAR_DOS_SEQ.Device.RVJ201_PID.PID_Enable := FALSE;                                      (* STEP: 95 *)
                               VAR_DOS_SEQ.Device.RVJ201_PID.PID_Mode := FALSE;
                               VAR_DOS_SEQ.Device.RVJ201_PID.Auto_SP_Value := 0;
                               VAR_DOS_SEQ.Device.RVJ201_PID.FIX_Value := 0;

                               VAR_DOS_SEQ.Device.AVJ201.AutoCnd := FALSE;                                             (* STEP: 95 Inlet Valve*)
                               VAR_DOS_SEQ.Device.AVJ201.EnableCnd := FALSE;
                               VAR_DOS_SEQ.Device.AVJ210.AutoCnd := FALSE;                                             (* STEP: 95 Washing Duct Valve*)
                               VAR_DOS_SEQ.Device.AVJ210.EnableCnd := FALSE;
                               VAR_DOS_SEQ.Device.AVJ211.AutoCnd := FALSE;                                             (* STEP: 95 Sprayball Valve*)
                               VAR_DOS_SEQ.Device.AVJ211.EnableCnd := FALSE;
                               VAR_DOS_SEQ.Device.AVJ212.AutoCnd := FALSE;                                             (* STEP: 95 *)
                               VAR_DOS_SEQ.Device.AVJ212.EnableCnd := FALSE;
                               VAR_DOS_SEQ.Device.AVJ215.AutoCnd := FALSE;                                             (* STEP: 95 Atmospheric drain valve*)
                               VAR_DOS_SEQ.Device.AVJ215.EnableCnd := FALSE;
                               VAR_DOS_SEQ.Device.AVJ216.AutoCnd := FALSE;                                             (* STEP: 95 Recirculation Valve*)
                               VAR_DOS_SEQ.Device.AVJ216.EnableCnd := FALSE;
                               VAR_DOS_SEQ.Device.AVJ217.AutoCnd := FALSE;                                             (* STEP: 95 Tank Hema Drain Valve*)
                               VAR_DOS_SEQ.Device.AVJ217.EnableCnd := FALSE;
                               VAR_DOS_SEQ.Device.AVJ218.AutoCnd := FALSE;                                             (* STEP: 95 Recirculation Valve*)
                               VAR_DOS_SEQ.Device.AVJ218.EnableCnd := FALSE;
                               VAR_DOS_SEQ.Device.AVJ221.AutoCnd := FALSE;                                             (* STEP: 95 Inlet Loop Valve*)
                               VAR_DOS_SEQ.Device.AVJ221.EnableCnd := FALSE;
                               VAR_DOS_SEQ.Device.AVJ230.AutoCnd := FALSE;                                             (* STEP: 95 *)
                               VAR_DOS_SEQ.Device.AVJ230.EnableCnd := FALSE;
                               VAR_DOS_SEQ.Device.AVJ231.AutoCnd := FALSE;                                             (* STEP: 95 *)
                               VAR_DOS_SEQ.Device.AVJ231.EnableCnd := FALSE;
                               VAR_DOS_SEQ.Device.AVJ232.AutoCnd := FALSE;                                             (* STEP: 95 *)
                               VAR_DOS_SEQ.Device.AVJ232.EnableCnd := FALSE;
                               VAR_DOS_SEQ.Device.AVJ233.AutoCnd := FALSE;                                             (* STEP: 95 *)
                               VAR_DOS_SEQ.Device.AVJ233.EnableCnd := FALSE;
                               VAR_DOS_SEQ.Device.AVJ234.AutoCnd := FALSE;                                             (* STEP: 95 *)
                               VAR_DOS_SEQ.Device.AVJ234.EnableCnd := FALSE;
                               VAR_DOS_SEQ.Device.AVJ235.AutoCnd := FALSE;                                             (* STEP: 95 *)
                               VAR_DOS_SEQ.Device.AVJ235.EnableCnd := FALSE;

                               VAR_DOS_SEQ.Device.LTJ203.ALR_HighLimitEn := FALSE;                                     (* STEP: 95 Hema Tank Level*)
                               VAR_DOS_SEQ.Device.LTJ203.ALR_HighLimitSP := 0;
                               VAR_DOS_SEQ.Device.LTJ203.ALR_LowLimitEn := FALSE;
                               VAR_DOS_SEQ.Device.LTJ203.ALR_LowLimitSP := 0;
                               VAR_DOS_SEQ.Device.LTJ203.SP := 0;
                               VAR_DOS_SEQ.Device.LTJ203.CMP := 0;
                               VAR_DOS_SEQ.Device.LTJ203.MinDev := 0;
                               VAR_DOS_SEQ.Device.LTJ203.MaxDev := 0;

                               VAR_DOS_SEQ.Device.TTJ203.ALR_HighLimitEn := FALSE;                                     (* STEP: 95 Hema Tank Temperature*)
                               VAR_DOS_SEQ.Device.TTJ203.ALR_HighLimitSP := 0;
                               VAR_DOS_SEQ.Device.TTJ203.ALR_LowLimitEn := FALSE;
                               VAR_DOS_SEQ.Device.TTJ203.ALR_LowLimitSP := 0;
                               VAR_DOS_SEQ.Device.TTJ203.SP := 0;
                               VAR_DOS_SEQ.Device.TTJ203.CMP := 0;
                               VAR_DOS_SEQ.Device.TTJ203.MinDev := 0;
                               VAR_DOS_SEQ.Device.TTJ203.MaxDev := 0;

                               VAR_DOS_SEQ.Device.LSJ200.ALR := FALSE;                                                 (* STEP: 95 *)
                               VAR_DOS_SEQ.Device.LSJ200.WAIT_OFF := FALSE;
                               VAR_DOS_SEQ.Device.LSJ200.WAIT_ON := FALSE;

                               VAR_DOS_SEQ.Device.LSJ201.ALR := FALSE;                                                 (* STEP: 95 *)
                               VAR_DOS_SEQ.Device.LSJ201.WAIT_OFF := FALSE;
                               VAR_DOS_SEQ.Device.LSJ201.WAIT_ON := FALSE;

                               VAR_DOS_SEQ.Device.LSJ202.ALR := FALSE;                                                 (* STEP: 95 *)
                               VAR_DOS_SEQ.Device.LSJ202.WAIT_OFF := FALSE;
                               VAR_DOS_SEQ.Device.LSJ202.WAIT_ON := FALSE;

                               VAR_DOS_SEQ.Device.FSJ201.ALR := FALSE;                                                 (* STEP: 95 *)
                               VAR_DOS_SEQ.Device.FSJ201.WAIT_OFF := FALSE;
                               VAR_DOS_SEQ.Device.FSJ201.WAIT_ON := FALSE;

                               VAR_DOS_SEQ.Device.FSJ202.ALR := FALSE;                                                 (* STEP: 95 *)
                               VAR_DOS_SEQ.Device.FSJ202.WAIT_OFF := FALSE;
                               VAR_DOS_SEQ.Device.FSJ202.WAIT_ON := FALSE;

                               VAR_DOS_SEQ.Mem.PBAbortEnable := TRUE;                                                  (* STEP: 95 PB Abort Sequence Enable*)
                               VAR_DOS_SEQ.Mem.PBStopEnable := FALSE;                                                  (* STEP: 95 PB Stop Sequence Enable*)
                               VAR_DOS_SEQ.Mem.PBStartEnable := FALSE;                                                 (* STEP: 95 PB Start Sequence Enable*)
                               VAR_DOS_SEQ.Mem.ContainersStop := TRUE;                                                 (* STEP: 95 *)
                               VAR_DOS_SEQ.Mem.MachineStart := FALSE;                                                  (* STEP: 95 *)
                               VAR_DOS_SEQ.Mem.MachineStop := TRUE;                                                    (* STEP: 95 *)
                               VAR_DOS_SEQ.Mem.DummyBottles := FALSE;                                                  (* STEP: 95 Dummy Bottle Install*)
                               VAR_DOS_SEQ.Mem.PositioningRequest := FALSE;                                            (* STEP: 95 Request of Cam Positioning at height SP of Sequncer*)
                               VAR_DOS_SEQ.Mem.COP_Cycle := FALSE;                                                     (* STEP: 95 COP Cycle Check Requested*)
                               VAR_DOS_SEQ.Mem.LapsCounter := FALSE;                                                   (* STEP: 95 *)
                               VAR_DOS_SEQ.Mem.ValveOpening := FALSE;                                                  (* STEP: 95 *)
                               VAR_DOS_SEQ.Mem.CopAfterCipRequest := FALSE;                                            (* STEP: 95 Request Of Cop After Cip*)

                               VAR_DOS_SEQ.ITC.CIP_CleaningRequest := FALSE;                                           (* STEP: 95 To CIP -> Request of Solution Sending*)
                               VAR_DOS_SEQ.ITC.CIP_Alarm := FALSE;                                                     (* STEP: 95 To CIP -> Critical Alarm Present*)
                               VAR_DOS_SEQ.ITC.CIP_RinseEnded := FALSE;                                                (* STEP: 95 To CIP -> Rinse Finished*)
                               VAR_DOS_SEQ.ITC.CIP_ChangeEnded := FALSE;                                               (* STEP: 95 To CIP -> Change Finished*)
                               VAR_DOS_SEQ.ITC.CIP_DrainRunning := FALSE;                                              (* STEP: 95 To CIP -> Drain Cycle Running*)
                               VAR_DOS_SEQ.ITC.CIP_RinseRunning := FALSE;                                              (* STEP: 95 To CIP -> Rinse Cycle Running*)
                               VAR_DOS_SEQ.ITC.CIP_CleaningRunning := FALSE;                                           (* STEP: 95 To CIP -> Cleaning Cycle Running*)
                               VAR_DOS_SEQ.ITC.CIP_DrainEnded := FALSE;                                                (* STEP: 95 To CIP -> Drain Finished*)
                               VAR_DOS_SEQ.ITC.CIP_FloodingEnded := FALSE;                                             (* STEP: 95 To CIP -> Flooding Finished*)
                               VAR_DOS_SEQ.ITC.CIP_FlipEnable := FALSE;                                                (* STEP: 95 *)
                               VAR_DOS_SEQ.ITC.CIP_CycleEnded := FALSE;                                                (* STEP: 95 *)

                               VAR_DOS_SEQ.ITC.PROD_ReadyForHeating := FALSE;                                          (* STEP: 95 To PASTO -> Filler Ready for Production (Heating)*)
                               VAR_DOS_SEQ.ITC.PROD_DoserInTemperature := FALSE;                                       (* STEP: 95 To PASTO -> Filler Temperature OK (After Heating)*)
                               VAR_DOS_SEQ.ITC.PROD_ProductRequest := FALSE;                                           (* STEP: 95 To PASTO -> Product Request*)
                               VAR_DOS_SEQ.ITC.PROD_DoserOnFillingMode := FALSE;                                       (* STEP: 95 To PASTO -> Product Consumend -Filling Valve Opening*)
                               VAR_DOS_SEQ.ITC.PROD_EndProductionCompleted := FALSE;                                   (* STEP: 95 To PASTO -> End Production Done*)
                               VAR_DOS_SEQ.ITC.PROD_ProductRecoveryEnd := FALSE;                                       (* STEP: 95 To PASTO -> Product Recovery End*)
                               VAR_DOS_SEQ.ITC.PROD_WaterRequestAfterProd := FALSE;                                    (* STEP: 95 To PASTO -> Water Request For Filler Rinse Afetr Production*)

                       96: (* C.I.P. -Press "STOP" to End the Cycle or Press "START" for a New Sequence *)

                               VAR_DOS_SEQ.Device.PPJ201_PID.PID_Enable := FALSE;                                      (* STEP: 96 Doser Recovery Pump*)
                               VAR_DOS_SEQ.Device.PPJ201_PID.PID_Mode := FALSE;
                               VAR_DOS_SEQ.Device.PPJ201_PID.Auto_SP_Value := 0;
                               VAR_DOS_SEQ.Device.PPJ201_PID.FIX_Value := 0;

                               VAR_DOS_SEQ.Device.PPJ202_PID.PID_Enable := FALSE;                                      (* STEP: 96 Doser Recovery Pump*)
                               VAR_DOS_SEQ.Device.PPJ202_PID.PID_Mode := FALSE;
                               VAR_DOS_SEQ.Device.PPJ202_PID.Auto_SP_Value := 0;
                               VAR_DOS_SEQ.Device.PPJ202_PID.FIX_Value := 0;

                               VAR_DOS_SEQ.Device.PPJ203_PID.PID_Enable := FALSE;                                      (* STEP: 96 Diaphragm Pump for Recovery pulp*)
                               VAR_DOS_SEQ.Device.PPJ203_PID.PID_Mode := FALSE;
                               VAR_DOS_SEQ.Device.PPJ203_PID.Auto_SP_Value := 0;
                               VAR_DOS_SEQ.Device.PPJ203_PID.FIX_Value := 0;

                               VAR_DOS_SEQ.Device.MMJ201_PID.PID_Enable := FALSE;                                      (* STEP: 96 Shaker Motor*)
                               VAR_DOS_SEQ.Device.MMJ201_PID.PID_Mode := FALSE;
                               VAR_DOS_SEQ.Device.MMJ201_PID.Auto_SP_Value := 0;
                               VAR_DOS_SEQ.Device.MMJ201_PID.FIX_Value := 0;

                               VAR_DOS_SEQ.Device.RVJ201_PID.PID_Enable := FALSE;                                      (* STEP: 96 *)
                               VAR_DOS_SEQ.Device.RVJ201_PID.PID_Mode := FALSE;
                               VAR_DOS_SEQ.Device.RVJ201_PID.Auto_SP_Value := 0;
                               VAR_DOS_SEQ.Device.RVJ201_PID.FIX_Value := 0;

                               VAR_DOS_SEQ.Device.AVJ201.AutoCnd := FALSE;                                             (* STEP: 96 Inlet Valve*)
                               VAR_DOS_SEQ.Device.AVJ201.EnableCnd := FALSE;
                               VAR_DOS_SEQ.Device.AVJ210.AutoCnd := FALSE;                                             (* STEP: 96 Washing Duct Valve*)
                               VAR_DOS_SEQ.Device.AVJ210.EnableCnd := FALSE;
                               VAR_DOS_SEQ.Device.AVJ211.AutoCnd := FALSE;                                             (* STEP: 96 Sprayball Valve*)
                               VAR_DOS_SEQ.Device.AVJ211.EnableCnd := FALSE;
                               VAR_DOS_SEQ.Device.AVJ212.AutoCnd := FALSE;                                             (* STEP: 96 *)
                               VAR_DOS_SEQ.Device.AVJ212.EnableCnd := FALSE;
                               VAR_DOS_SEQ.Device.AVJ215.AutoCnd := FALSE;                                             (* STEP: 96 Atmospheric drain valve*)
                               VAR_DOS_SEQ.Device.AVJ215.EnableCnd := FALSE;
                               VAR_DOS_SEQ.Device.AVJ216.AutoCnd := FALSE;                                             (* STEP: 96 Recirculation Valve*)
                               VAR_DOS_SEQ.Device.AVJ216.EnableCnd := FALSE;
                               VAR_DOS_SEQ.Device.AVJ217.AutoCnd := FALSE;                                             (* STEP: 96 Tank Hema Drain Valve*)
                               VAR_DOS_SEQ.Device.AVJ217.EnableCnd := FALSE;
                               VAR_DOS_SEQ.Device.AVJ218.AutoCnd := FALSE;                                             (* STEP: 96 Recirculation Valve*)
                               VAR_DOS_SEQ.Device.AVJ218.EnableCnd := FALSE;
                               VAR_DOS_SEQ.Device.AVJ221.AutoCnd := FALSE;                                             (* STEP: 96 Inlet Loop Valve*)
                               VAR_DOS_SEQ.Device.AVJ221.EnableCnd := FALSE;
                               VAR_DOS_SEQ.Device.AVJ230.AutoCnd := FALSE;                                             (* STEP: 96 *)
                               VAR_DOS_SEQ.Device.AVJ230.EnableCnd := FALSE;
                               VAR_DOS_SEQ.Device.AVJ231.AutoCnd := FALSE;                                             (* STEP: 96 *)
                               VAR_DOS_SEQ.Device.AVJ231.EnableCnd := FALSE;
                               VAR_DOS_SEQ.Device.AVJ232.AutoCnd := FALSE;                                             (* STEP: 96 *)
                               VAR_DOS_SEQ.Device.AVJ232.EnableCnd := FALSE;
                               VAR_DOS_SEQ.Device.AVJ233.AutoCnd := FALSE;                                             (* STEP: 96 *)
                               VAR_DOS_SEQ.Device.AVJ233.EnableCnd := FALSE;
                               VAR_DOS_SEQ.Device.AVJ234.AutoCnd := FALSE;                                             (* STEP: 96 *)
                               VAR_DOS_SEQ.Device.AVJ234.EnableCnd := FALSE;
                               VAR_DOS_SEQ.Device.AVJ235.AutoCnd := FALSE;                                             (* STEP: 96 *)
                               VAR_DOS_SEQ.Device.AVJ235.EnableCnd := FALSE;

                               VAR_DOS_SEQ.Device.LTJ203.ALR_HighLimitEn := FALSE;                                     (* STEP: 96 Hema Tank Level*)
                               VAR_DOS_SEQ.Device.LTJ203.ALR_HighLimitSP := 0;
                               VAR_DOS_SEQ.Device.LTJ203.ALR_LowLimitEn := FALSE;
                               VAR_DOS_SEQ.Device.LTJ203.ALR_LowLimitSP := 0;
                               VAR_DOS_SEQ.Device.LTJ203.SP := 0;
                               VAR_DOS_SEQ.Device.LTJ203.CMP := 0;
                               VAR_DOS_SEQ.Device.LTJ203.MinDev := 0;
                               VAR_DOS_SEQ.Device.LTJ203.MaxDev := 0;

                               VAR_DOS_SEQ.Device.TTJ203.ALR_HighLimitEn := FALSE;                                     (* STEP: 96 Hema Tank Temperature*)
                               VAR_DOS_SEQ.Device.TTJ203.ALR_HighLimitSP := 0;
                               VAR_DOS_SEQ.Device.TTJ203.ALR_LowLimitEn := FALSE;
                               VAR_DOS_SEQ.Device.TTJ203.ALR_LowLimitSP := 0;
                               VAR_DOS_SEQ.Device.TTJ203.SP := 0;
                               VAR_DOS_SEQ.Device.TTJ203.CMP := 0;
                               VAR_DOS_SEQ.Device.TTJ203.MinDev := 0;
                               VAR_DOS_SEQ.Device.TTJ203.MaxDev := 0;

                               VAR_DOS_SEQ.Device.LSJ200.ALR := FALSE;                                                 (* STEP: 96 *)
                               VAR_DOS_SEQ.Device.LSJ200.WAIT_OFF := FALSE;
                               VAR_DOS_SEQ.Device.LSJ200.WAIT_ON := FALSE;

                               VAR_DOS_SEQ.Device.LSJ201.ALR := FALSE;                                                 (* STEP: 96 *)
                               VAR_DOS_SEQ.Device.LSJ201.WAIT_OFF := FALSE;
                               VAR_DOS_SEQ.Device.LSJ201.WAIT_ON := FALSE;

                               VAR_DOS_SEQ.Device.LSJ202.ALR := FALSE;                                                 (* STEP: 96 *)
                               VAR_DOS_SEQ.Device.LSJ202.WAIT_OFF := FALSE;
                               VAR_DOS_SEQ.Device.LSJ202.WAIT_ON := FALSE;

                               VAR_DOS_SEQ.Device.FSJ201.ALR := FALSE;                                                 (* STEP: 96 *)
                               VAR_DOS_SEQ.Device.FSJ201.WAIT_OFF := FALSE;
                               VAR_DOS_SEQ.Device.FSJ201.WAIT_ON := FALSE;

                               VAR_DOS_SEQ.Device.FSJ202.ALR := FALSE;                                                 (* STEP: 96 *)
                               VAR_DOS_SEQ.Device.FSJ202.WAIT_OFF := FALSE;
                               VAR_DOS_SEQ.Device.FSJ202.WAIT_ON := FALSE;

                               VAR_DOS_SEQ.Mem.PBAbortEnable := FALSE;                                                 (* STEP: 96 PB Abort Sequence Enable*)
                               VAR_DOS_SEQ.Mem.PBStopEnable := TRUE;                                                   (* STEP: 96 PB Stop Sequence Enable*)
                               VAR_DOS_SEQ.Mem.PBStartEnable := TRUE;                                                  (* STEP: 96 PB Start Sequence Enable*)
                               VAR_DOS_SEQ.Mem.ContainersStop := FALSE;                                                (* STEP: 96 *)
                               VAR_DOS_SEQ.Mem.MachineStart := FALSE;                                                  (* STEP: 96 *)
                               VAR_DOS_SEQ.Mem.MachineStop := TRUE;                                                    (* STEP: 96 *)
                               VAR_DOS_SEQ.Mem.DummyBottles := FALSE;                                                  (* STEP: 96 Dummy Bottle Install*)
                               VAR_DOS_SEQ.Mem.PositioningRequest := FALSE;                                            (* STEP: 96 Request of Cam Positioning at height SP of Sequncer*)
                               VAR_DOS_SEQ.Mem.COP_Cycle := FALSE;                                                     (* STEP: 96 COP Cycle Check Requested*)
                               VAR_DOS_SEQ.Mem.LapsCounter := FALSE;                                                   (* STEP: 96 *)
                               VAR_DOS_SEQ.Mem.ValveOpening := FALSE;                                                  (* STEP: 96 *)
                               VAR_DOS_SEQ.Mem.CopAfterCipRequest := FALSE;                                            (* STEP: 96 Request Of Cop After Cip*)

                               VAR_DOS_SEQ.ITC.CIP_CleaningRequest := FALSE;                                           (* STEP: 96 To CIP -> Request of Solution Sending*)
                               VAR_DOS_SEQ.ITC.CIP_Alarm := FALSE;                                                     (* STEP: 96 To CIP -> Critical Alarm Present*)
                               VAR_DOS_SEQ.ITC.CIP_RinseEnded := FALSE;                                                (* STEP: 96 To CIP -> Rinse Finished*)
                               VAR_DOS_SEQ.ITC.CIP_ChangeEnded := FALSE;                                               (* STEP: 96 To CIP -> Change Finished*)
                               VAR_DOS_SEQ.ITC.CIP_DrainRunning := FALSE;                                              (* STEP: 96 To CIP -> Drain Cycle Running*)
                               VAR_DOS_SEQ.ITC.CIP_RinseRunning := FALSE;                                              (* STEP: 96 To CIP -> Rinse Cycle Running*)
                               VAR_DOS_SEQ.ITC.CIP_CleaningRunning := FALSE;                                           (* STEP: 96 To CIP -> Cleaning Cycle Running*)
                               VAR_DOS_SEQ.ITC.CIP_DrainEnded := FALSE;                                                (* STEP: 96 To CIP -> Drain Finished*)
                               VAR_DOS_SEQ.ITC.CIP_FloodingEnded := FALSE;                                             (* STEP: 96 To CIP -> Flooding Finished*)
                               VAR_DOS_SEQ.ITC.CIP_FlipEnable := FALSE;                                                (* STEP: 96 *)
                               VAR_DOS_SEQ.ITC.CIP_CycleEnded := FALSE;                                                (* STEP: 96 *)

                               VAR_DOS_SEQ.ITC.PROD_ReadyForHeating := FALSE;                                          (* STEP: 96 To PASTO -> Filler Ready for Production (Heating)*)
                               VAR_DOS_SEQ.ITC.PROD_DoserInTemperature := FALSE;                                       (* STEP: 96 To PASTO -> Filler Temperature OK (After Heating)*)
                               VAR_DOS_SEQ.ITC.PROD_ProductRequest := FALSE;                                           (* STEP: 96 To PASTO -> Product Request*)
                               VAR_DOS_SEQ.ITC.PROD_DoserOnFillingMode := FALSE;                                       (* STEP: 96 To PASTO -> Product Consumend -Filling Valve Opening*)
                               VAR_DOS_SEQ.ITC.PROD_EndProductionCompleted := FALSE;                                   (* STEP: 96 To PASTO -> End Production Done*)
                               VAR_DOS_SEQ.ITC.PROD_ProductRecoveryEnd := FALSE;                                       (* STEP: 96 To PASTO -> Product Recovery End*)
                               VAR_DOS_SEQ.ITC.PROD_WaterRequestAfterProd := FALSE;                                    (* STEP: 96 To PASTO -> Water Request For Filler Rinse Afetr Production*)

                       97..99: (* Spare Steps *)

                       100: (* RINSE -Tank Emptying *)

                               VAR_DOS_SEQ.Device.PPJ201_PID.PID_Enable := FALSE;                                      (* STEP: 100 Doser Recovery Pump*)
                               VAR_DOS_SEQ.Device.PPJ201_PID.PID_Mode := FALSE;
                               VAR_DOS_SEQ.Device.PPJ201_PID.Auto_SP_Value := 0;
                               VAR_DOS_SEQ.Device.PPJ201_PID.FIX_Value := 0;

                               VAR_DOS_SEQ.Device.PPJ202_PID.PID_Enable := FALSE;                                      (* STEP: 100 Doser Recovery Pump*)
                               VAR_DOS_SEQ.Device.PPJ202_PID.PID_Mode := FALSE;
                               VAR_DOS_SEQ.Device.PPJ202_PID.Auto_SP_Value := 0;
                               VAR_DOS_SEQ.Device.PPJ202_PID.FIX_Value := 0;

                               VAR_DOS_SEQ.Device.PPJ203_PID.PID_Enable := FALSE;                                      (* STEP: 100 Diaphragm Pump for Recovery pulp*)
                               VAR_DOS_SEQ.Device.PPJ203_PID.PID_Mode := FALSE;
                               VAR_DOS_SEQ.Device.PPJ203_PID.Auto_SP_Value := 0;
                               VAR_DOS_SEQ.Device.PPJ203_PID.FIX_Value := 0;

                               VAR_DOS_SEQ.Device.MMJ201_PID.PID_Enable := FALSE;                                      (* STEP: 100 Shaker Motor*)
                               VAR_DOS_SEQ.Device.MMJ201_PID.PID_Mode := FALSE;
                               VAR_DOS_SEQ.Device.MMJ201_PID.Auto_SP_Value := 0;
                               VAR_DOS_SEQ.Device.MMJ201_PID.FIX_Value := 0;

                               VAR_DOS_SEQ.Device.RVJ201_PID.PID_Enable := FALSE;                                      (* STEP: 100 *)
                               VAR_DOS_SEQ.Device.RVJ201_PID.PID_Mode := FALSE;
                               VAR_DOS_SEQ.Device.RVJ201_PID.Auto_SP_Value := 0;
                               VAR_DOS_SEQ.Device.RVJ201_PID.FIX_Value := 0;

                               VAR_DOS_SEQ.Device.AVJ201.AutoCnd := FALSE;                                             (* STEP: 100 Inlet Valve*)
                               VAR_DOS_SEQ.Device.AVJ201.EnableCnd := FALSE;
                               VAR_DOS_SEQ.Device.AVJ210.AutoCnd := FALSE;                                             (* STEP: 100 Washing Duct Valve*)
                               VAR_DOS_SEQ.Device.AVJ210.EnableCnd := FALSE;
                               VAR_DOS_SEQ.Device.AVJ211.AutoCnd := FALSE;                                             (* STEP: 100 Sprayball Valve*)
                               VAR_DOS_SEQ.Device.AVJ211.EnableCnd := FALSE;
                               VAR_DOS_SEQ.Device.AVJ212.AutoCnd := FALSE;                                             (* STEP: 100 *)
                               VAR_DOS_SEQ.Device.AVJ212.EnableCnd := FALSE;
                               VAR_DOS_SEQ.Device.AVJ215.AutoCnd := TRUE;                                              (* STEP: 100 Atmospheric drain valve*)
                               VAR_DOS_SEQ.Device.AVJ215.EnableCnd := FALSE;
                               VAR_DOS_SEQ.Device.AVJ216.AutoCnd := FALSE;                                             (* STEP: 100 Recirculation Valve*)
                               VAR_DOS_SEQ.Device.AVJ216.EnableCnd := FALSE;
                               VAR_DOS_SEQ.Device.AVJ217.AutoCnd := TRUE;                                              (* STEP: 100 Tank Hema Drain Valve*)
                               VAR_DOS_SEQ.Device.AVJ217.EnableCnd := FALSE;
                               VAR_DOS_SEQ.Device.AVJ218.AutoCnd := FALSE;                                             (* STEP: 100 Recirculation Valve*)
                               VAR_DOS_SEQ.Device.AVJ218.EnableCnd := FALSE;
                               VAR_DOS_SEQ.Device.AVJ221.AutoCnd := FALSE;                                             (* STEP: 100 Inlet Loop Valve*)
                               VAR_DOS_SEQ.Device.AVJ221.EnableCnd := FALSE;
                               VAR_DOS_SEQ.Device.AVJ230.AutoCnd := FALSE;                                             (* STEP: 100 *)
                               VAR_DOS_SEQ.Device.AVJ230.EnableCnd := FALSE;
                               VAR_DOS_SEQ.Device.AVJ231.AutoCnd := FALSE;                                             (* STEP: 100 *)
                               VAR_DOS_SEQ.Device.AVJ231.EnableCnd := FALSE;
                               VAR_DOS_SEQ.Device.AVJ232.AutoCnd := TRUE;                                              (* STEP: 100 *)
                               VAR_DOS_SEQ.Device.AVJ232.EnableCnd := FALSE;
                               VAR_DOS_SEQ.Device.AVJ233.AutoCnd := FALSE;                                             (* STEP: 100 *)
                               VAR_DOS_SEQ.Device.AVJ233.EnableCnd := FALSE;
                               VAR_DOS_SEQ.Device.AVJ234.AutoCnd := FALSE;                                             (* STEP: 100 *)
                               VAR_DOS_SEQ.Device.AVJ234.EnableCnd := FALSE;
                               VAR_DOS_SEQ.Device.AVJ235.AutoCnd := FALSE;                                             (* STEP: 100 *)
                               VAR_DOS_SEQ.Device.AVJ235.EnableCnd := FALSE;

                               VAR_DOS_SEQ.Device.LTJ203.ALR_HighLimitEn := FALSE;                                     (* STEP: 100 Hema Tank Level*)
                               VAR_DOS_SEQ.Device.LTJ203.ALR_HighLimitSP := 0;
                               VAR_DOS_SEQ.Device.LTJ203.ALR_LowLimitEn := FALSE;
                               VAR_DOS_SEQ.Device.LTJ203.ALR_LowLimitSP := 0;
                               VAR_DOS_SEQ.Device.LTJ203.SP := 5;
                               VAR_DOS_SEQ.Device.LTJ203.CMP := 1;
                               VAR_DOS_SEQ.Device.LTJ203.MinDev := 0;
                               VAR_DOS_SEQ.Device.LTJ203.MaxDev := 0;

                               VAR_DOS_SEQ.Device.TTJ203.ALR_HighLimitEn := FALSE;                                     (* STEP: 100 Hema Tank Temperature*)
                               VAR_DOS_SEQ.Device.TTJ203.ALR_HighLimitSP := 0;
                               VAR_DOS_SEQ.Device.TTJ203.ALR_LowLimitEn := FALSE;
                               VAR_DOS_SEQ.Device.TTJ203.ALR_LowLimitSP := 0;
                               VAR_DOS_SEQ.Device.TTJ203.SP := 0;
                               VAR_DOS_SEQ.Device.TTJ203.CMP := 0;
                               VAR_DOS_SEQ.Device.TTJ203.MinDev := 0;
                               VAR_DOS_SEQ.Device.TTJ203.MaxDev := 0;

                               VAR_DOS_SEQ.Device.LSJ200.ALR := FALSE;                                                 (* STEP: 100 *)
                               VAR_DOS_SEQ.Device.LSJ200.WAIT_OFF := FALSE;
                               VAR_DOS_SEQ.Device.LSJ200.WAIT_ON := FALSE;

                               VAR_DOS_SEQ.Device.LSJ201.ALR := FALSE;                                                 (* STEP: 100 *)
                               VAR_DOS_SEQ.Device.LSJ201.WAIT_OFF := FALSE;
                               VAR_DOS_SEQ.Device.LSJ201.WAIT_ON := FALSE;

                               VAR_DOS_SEQ.Device.LSJ202.ALR := FALSE;                                                 (* STEP: 100 *)
                               VAR_DOS_SEQ.Device.LSJ202.WAIT_OFF := FALSE;
                               VAR_DOS_SEQ.Device.LSJ202.WAIT_ON := FALSE;

                               VAR_DOS_SEQ.Device.FSJ201.ALR := FALSE;                                                 (* STEP: 100 *)
                               VAR_DOS_SEQ.Device.FSJ201.WAIT_OFF := FALSE;
                               VAR_DOS_SEQ.Device.FSJ201.WAIT_ON := FALSE;

                               VAR_DOS_SEQ.Device.FSJ202.ALR := FALSE;                                                 (* STEP: 100 *)
                               VAR_DOS_SEQ.Device.FSJ202.WAIT_OFF := FALSE;
                               VAR_DOS_SEQ.Device.FSJ202.WAIT_ON := FALSE;

                               VAR_DOS_SEQ.Mem.PBAbortEnable := TRUE;                                                  (* STEP: 100 PB Abort Sequence Enable*)
                               VAR_DOS_SEQ.Mem.PBStopEnable := TRUE;                                                   (* STEP: 100 PB Stop Sequence Enable*)
                               VAR_DOS_SEQ.Mem.PBStartEnable := FALSE;                                                 (* STEP: 100 PB Start Sequence Enable*)
                               VAR_DOS_SEQ.Mem.ContainersStop := TRUE;                                                 (* STEP: 100 *)
                               VAR_DOS_SEQ.Mem.MachineStart := FALSE;                                                  (* STEP: 100 *)
                               VAR_DOS_SEQ.Mem.MachineStop := FALSE;                                                   (* STEP: 100 *)
                               VAR_DOS_SEQ.Mem.DummyBottles := FALSE;                                                  (* STEP: 100 Dummy Bottle Install*)
                               VAR_DOS_SEQ.Mem.PositioningRequest := FALSE;                                            (* STEP: 100 Request of Cam Positioning at height SP of Sequncer*)
                               VAR_DOS_SEQ.Mem.COP_Cycle := FALSE;                                                     (* STEP: 100 COP Cycle Check Requested*)
                               VAR_DOS_SEQ.Mem.LapsCounter := FALSE;                                                   (* STEP: 100 *)
                               VAR_DOS_SEQ.Mem.ValveOpening := FALSE;                                                  (* STEP: 100 *)
                               VAR_DOS_SEQ.Mem.CopAfterCipRequest := FALSE;                                            (* STEP: 100 Request Of Cop After Cip*)

                               VAR_DOS_SEQ.ITC.CIP_CleaningRequest := FALSE;                                           (* STEP: 100 To CIP -> Request of Solution Sending*)
                               VAR_DOS_SEQ.ITC.CIP_Alarm := FALSE;                                                     (* STEP: 100 To CIP -> Critical Alarm Present*)
                               VAR_DOS_SEQ.ITC.CIP_RinseEnded := FALSE;                                                (* STEP: 100 To CIP -> Rinse Finished*)
                               VAR_DOS_SEQ.ITC.CIP_ChangeEnded := FALSE;                                               (* STEP: 100 To CIP -> Change Finished*)
                               VAR_DOS_SEQ.ITC.CIP_DrainRunning := FALSE;                                              (* STEP: 100 To CIP -> Drain Cycle Running*)
                               VAR_DOS_SEQ.ITC.CIP_RinseRunning := TRUE;                                               (* STEP: 100 To CIP -> Rinse Cycle Running*)
                               VAR_DOS_SEQ.ITC.CIP_CleaningRunning := FALSE;                                           (* STEP: 100 To CIP -> Cleaning Cycle Running*)
                               VAR_DOS_SEQ.ITC.CIP_DrainEnded := FALSE;                                                (* STEP: 100 To CIP -> Drain Finished*)
                               VAR_DOS_SEQ.ITC.CIP_FloodingEnded := FALSE;                                             (* STEP: 100 To CIP -> Flooding Finished*)
                               VAR_DOS_SEQ.ITC.CIP_FlipEnable := FALSE;                                                (* STEP: 100 *)
                               VAR_DOS_SEQ.ITC.CIP_CycleEnded := FALSE;                                                (* STEP: 100 *)

                               VAR_DOS_SEQ.ITC.PROD_ReadyForHeating := FALSE;                                          (* STEP: 100 To PASTO -> Filler Ready for Production (Heating)*)
                               VAR_DOS_SEQ.ITC.PROD_DoserInTemperature := FALSE;                                       (* STEP: 100 To PASTO -> Filler Temperature OK (After Heating)*)
                               VAR_DOS_SEQ.ITC.PROD_ProductRequest := FALSE;                                           (* STEP: 100 To PASTO -> Product Request*)
                               VAR_DOS_SEQ.ITC.PROD_DoserOnFillingMode := FALSE;                                       (* STEP: 100 To PASTO -> Product Consumend -Filling Valve Opening*)
                               VAR_DOS_SEQ.ITC.PROD_EndProductionCompleted := FALSE;                                   (* STEP: 100 To PASTO -> End Production Done*)
                               VAR_DOS_SEQ.ITC.PROD_ProductRecoveryEnd := FALSE;                                       (* STEP: 100 To PASTO -> Product Recovery End*)
                               VAR_DOS_SEQ.ITC.PROD_WaterRequestAfterProd := FALSE;                                    (* STEP: 100 To PASTO -> Water Request For Filler Rinse Afetr Production*)

                       101: (* RINSE -Rinse Product Pipes *)

                               VAR_DOS_SEQ.Device.PPJ201_PID.PID_Enable := FALSE;                                      (* STEP: 101 Doser Recovery Pump*)
                               VAR_DOS_SEQ.Device.PPJ201_PID.PID_Mode := FALSE;
                               VAR_DOS_SEQ.Device.PPJ201_PID.Auto_SP_Value := 0;
                               VAR_DOS_SEQ.Device.PPJ201_PID.FIX_Value := 0;

                               VAR_DOS_SEQ.Device.PPJ202_PID.PID_Enable := FALSE;                                      (* STEP: 101 Doser Recovery Pump*)
                               VAR_DOS_SEQ.Device.PPJ202_PID.PID_Mode := FALSE;
                               VAR_DOS_SEQ.Device.PPJ202_PID.Auto_SP_Value := 0;
                               VAR_DOS_SEQ.Device.PPJ202_PID.FIX_Value := 0;

                               VAR_DOS_SEQ.Device.PPJ203_PID.PID_Enable := FALSE;                                      (* STEP: 101 Diaphragm Pump for Recovery pulp*)
                               VAR_DOS_SEQ.Device.PPJ203_PID.PID_Mode := FALSE;
                               VAR_DOS_SEQ.Device.PPJ203_PID.Auto_SP_Value := 0;
                               VAR_DOS_SEQ.Device.PPJ203_PID.FIX_Value := 0;

                               VAR_DOS_SEQ.Device.MMJ201_PID.PID_Enable := TRUE;                                       (* STEP: 101 Shaker Motor*)
                               VAR_DOS_SEQ.Device.MMJ201_PID.PID_Mode := TRUE;
                               VAR_DOS_SEQ.Device.MMJ201_PID.Auto_SP_Value := 10;
                               VAR_DOS_SEQ.Device.MMJ201_PID.FIX_Value := 0;

                               VAR_DOS_SEQ.Device.RVJ201_PID.PID_Enable := FALSE;                                      (* STEP: 101 *)
                               VAR_DOS_SEQ.Device.RVJ201_PID.PID_Mode := FALSE;
                               VAR_DOS_SEQ.Device.RVJ201_PID.Auto_SP_Value := 0;
                               VAR_DOS_SEQ.Device.RVJ201_PID.FIX_Value := 0;

                               VAR_DOS_SEQ.Device.AVJ201.AutoCnd := TRUE;                                              (* STEP: 101 Inlet Valve*)
                               VAR_DOS_SEQ.Device.AVJ201.EnableCnd := TRUE;
                               VAR_DOS_SEQ.Device.AVJ210.AutoCnd := FALSE;                                             (* STEP: 101 Washing Duct Valve*)
                               VAR_DOS_SEQ.Device.AVJ210.EnableCnd := FALSE;
                               VAR_DOS_SEQ.Device.AVJ211.AutoCnd := FALSE;                                             (* STEP: 101 Sprayball Valve*)
                               VAR_DOS_SEQ.Device.AVJ211.EnableCnd := FALSE;
                               VAR_DOS_SEQ.Device.AVJ212.AutoCnd := FALSE;                                             (* STEP: 101 *)
                               VAR_DOS_SEQ.Device.AVJ212.EnableCnd := FALSE;
                               VAR_DOS_SEQ.Device.AVJ215.AutoCnd := TRUE;                                              (* STEP: 101 Atmospheric drain valve*)
                               VAR_DOS_SEQ.Device.AVJ215.EnableCnd := FALSE;
                               VAR_DOS_SEQ.Device.AVJ216.AutoCnd := FALSE;                                             (* STEP: 101 Recirculation Valve*)
                               VAR_DOS_SEQ.Device.AVJ216.EnableCnd := FALSE;
                               VAR_DOS_SEQ.Device.AVJ217.AutoCnd := TRUE;                                              (* STEP: 101 Tank Hema Drain Valve*)
                               VAR_DOS_SEQ.Device.AVJ217.EnableCnd := FALSE;
                               VAR_DOS_SEQ.Device.AVJ218.AutoCnd := FALSE;                                             (* STEP: 101 Recirculation Valve*)
                               VAR_DOS_SEQ.Device.AVJ218.EnableCnd := FALSE;
                               VAR_DOS_SEQ.Device.AVJ221.AutoCnd := FALSE;                                             (* STEP: 101 Inlet Loop Valve*)
                               VAR_DOS_SEQ.Device.AVJ221.EnableCnd := FALSE;
                               VAR_DOS_SEQ.Device.AVJ230.AutoCnd := TRUE;                                              (* STEP: 101 *)
                               VAR_DOS_SEQ.Device.AVJ230.EnableCnd := FALSE;
                               VAR_DOS_SEQ.Device.AVJ231.AutoCnd := FALSE;                                             (* STEP: 101 *)
                               VAR_DOS_SEQ.Device.AVJ231.EnableCnd := FALSE;
                               VAR_DOS_SEQ.Device.AVJ232.AutoCnd := TRUE;                                              (* STEP: 101 *)
                               VAR_DOS_SEQ.Device.AVJ232.EnableCnd := FALSE;
                               VAR_DOS_SEQ.Device.AVJ233.AutoCnd := FALSE;                                             (* STEP: 101 *)
                               VAR_DOS_SEQ.Device.AVJ233.EnableCnd := FALSE;
                               VAR_DOS_SEQ.Device.AVJ234.AutoCnd := TRUE;                                              (* STEP: 101 *)
                               VAR_DOS_SEQ.Device.AVJ234.EnableCnd := FALSE;
                               VAR_DOS_SEQ.Device.AVJ235.AutoCnd := FALSE;                                             (* STEP: 101 *)
                               VAR_DOS_SEQ.Device.AVJ235.EnableCnd := FALSE;

                               VAR_DOS_SEQ.Device.LTJ203.ALR_HighLimitEn := TRUE;                                      (* STEP: 101 Hema Tank Level*)
                               VAR_DOS_SEQ.Device.LTJ203.ALR_HighLimitSP := HMI_PAM_3._607;
                               VAR_DOS_SEQ.Device.LTJ203.ALR_LowLimitEn := TRUE;
                               VAR_DOS_SEQ.Device.LTJ203.ALR_LowLimitSP := HMI_PAM_3._606;
                               VAR_DOS_SEQ.Device.LTJ203.SP := HMI_PAM_3._626;
                               VAR_DOS_SEQ.Device.LTJ203.CMP := 2;
                               VAR_DOS_SEQ.Device.LTJ203.MinDev := 0;
                               VAR_DOS_SEQ.Device.LTJ203.MaxDev := 0;

                               VAR_DOS_SEQ.Device.TTJ203.ALR_HighLimitEn := FALSE;                                     (* STEP: 101 Hema Tank Temperature*)
                               VAR_DOS_SEQ.Device.TTJ203.ALR_HighLimitSP := 0;
                               VAR_DOS_SEQ.Device.TTJ203.ALR_LowLimitEn := FALSE;
                               VAR_DOS_SEQ.Device.TTJ203.ALR_LowLimitSP := 0;
                               VAR_DOS_SEQ.Device.TTJ203.SP := 0;
                               VAR_DOS_SEQ.Device.TTJ203.CMP := 0;
                               VAR_DOS_SEQ.Device.TTJ203.MinDev := 0;
                               VAR_DOS_SEQ.Device.TTJ203.MaxDev := 0;

                               VAR_DOS_SEQ.Device.LSJ200.ALR := FALSE;                                                 (* STEP: 101 *)
                               VAR_DOS_SEQ.Device.LSJ200.WAIT_OFF := FALSE;
                               VAR_DOS_SEQ.Device.LSJ200.WAIT_ON := FALSE;

                               VAR_DOS_SEQ.Device.LSJ201.ALR := FALSE;                                                 (* STEP: 101 *)
                               VAR_DOS_SEQ.Device.LSJ201.WAIT_OFF := FALSE;
                               VAR_DOS_SEQ.Device.LSJ201.WAIT_ON := FALSE;

                               VAR_DOS_SEQ.Device.LSJ202.ALR := FALSE;                                                 (* STEP: 101 *)
                               VAR_DOS_SEQ.Device.LSJ202.WAIT_OFF := FALSE;
                               VAR_DOS_SEQ.Device.LSJ202.WAIT_ON := FALSE;

                               VAR_DOS_SEQ.Device.FSJ201.ALR := FALSE;                                                 (* STEP: 101 *)
                               VAR_DOS_SEQ.Device.FSJ201.WAIT_OFF := FALSE;
                               VAR_DOS_SEQ.Device.FSJ201.WAIT_ON := FALSE;

                               VAR_DOS_SEQ.Device.FSJ202.ALR := FALSE;                                                 (* STEP: 101 *)
                               VAR_DOS_SEQ.Device.FSJ202.WAIT_OFF := FALSE;
                               VAR_DOS_SEQ.Device.FSJ202.WAIT_ON := FALSE;

                               VAR_DOS_SEQ.Mem.PBAbortEnable := TRUE;                                                  (* STEP: 101 PB Abort Sequence Enable*)
                               VAR_DOS_SEQ.Mem.PBStopEnable := TRUE;                                                   (* STEP: 101 PB Stop Sequence Enable*)
                               VAR_DOS_SEQ.Mem.PBStartEnable := FALSE;                                                 (* STEP: 101 PB Start Sequence Enable*)
                               VAR_DOS_SEQ.Mem.ContainersStop := TRUE;                                                 (* STEP: 101 *)
                               VAR_DOS_SEQ.Mem.MachineStart := TRUE;                                                   (* STEP: 101 *)
                               VAR_DOS_SEQ.Mem.MachineStop := FALSE;                                                   (* STEP: 101 *)
                               VAR_DOS_SEQ.Mem.DummyBottles := FALSE;                                                  (* STEP: 101 Dummy Bottle Install*)
                               VAR_DOS_SEQ.Mem.PositioningRequest := FALSE;                                            (* STEP: 101 Request of Cam Positioning at height SP of Sequncer*)
                               VAR_DOS_SEQ.Mem.COP_Cycle := FALSE;                                                     (* STEP: 101 COP Cycle Check Requested*)
                               VAR_DOS_SEQ.Mem.LapsCounter := FALSE;                                                   (* STEP: 101 *)
                               VAR_DOS_SEQ.Mem.ValveOpening := FALSE;                                                  (* STEP: 101 *)
                               VAR_DOS_SEQ.Mem.CopAfterCipRequest := FALSE;                                            (* STEP: 101 Request Of Cop After Cip*)

                               VAR_DOS_SEQ.ITC.CIP_CleaningRequest := FALSE;                                           (* STEP: 101 To CIP -> Request of Solution Sending*)
                               VAR_DOS_SEQ.ITC.CIP_Alarm := FALSE;                                                     (* STEP: 101 To CIP -> Critical Alarm Present*)
                               VAR_DOS_SEQ.ITC.CIP_RinseEnded := FALSE;                                                (* STEP: 101 To CIP -> Rinse Finished*)
                               VAR_DOS_SEQ.ITC.CIP_ChangeEnded := FALSE;                                               (* STEP: 101 To CIP -> Change Finished*)
                               VAR_DOS_SEQ.ITC.CIP_DrainRunning := FALSE;                                              (* STEP: 101 To CIP -> Drain Cycle Running*)
                               VAR_DOS_SEQ.ITC.CIP_RinseRunning := TRUE;                                               (* STEP: 101 To CIP -> Rinse Cycle Running*)
                               VAR_DOS_SEQ.ITC.CIP_CleaningRunning := FALSE;                                           (* STEP: 101 To CIP -> Cleaning Cycle Running*)
                               VAR_DOS_SEQ.ITC.CIP_DrainEnded := FALSE;                                                (* STEP: 101 To CIP -> Drain Finished*)
                               VAR_DOS_SEQ.ITC.CIP_FloodingEnded := FALSE;                                             (* STEP: 101 To CIP -> Flooding Finished*)
                               VAR_DOS_SEQ.ITC.CIP_FlipEnable := FALSE;                                                (* STEP: 101 *)
                               VAR_DOS_SEQ.ITC.CIP_CycleEnded := FALSE;                                                (* STEP: 101 *)

                               VAR_DOS_SEQ.ITC.PROD_ReadyForHeating := FALSE;                                          (* STEP: 101 To PASTO -> Filler Ready for Production (Heating)*)
                               VAR_DOS_SEQ.ITC.PROD_DoserInTemperature := FALSE;                                       (* STEP: 101 To PASTO -> Filler Temperature OK (After Heating)*)
                               VAR_DOS_SEQ.ITC.PROD_ProductRequest := FALSE;                                           (* STEP: 101 To PASTO -> Product Request*)
                               VAR_DOS_SEQ.ITC.PROD_DoserOnFillingMode := FALSE;                                       (* STEP: 101 To PASTO -> Product Consumend -Filling Valve Opening*)
                               VAR_DOS_SEQ.ITC.PROD_EndProductionCompleted := FALSE;                                   (* STEP: 101 To PASTO -> End Production Done*)
                               VAR_DOS_SEQ.ITC.PROD_ProductRecoveryEnd := FALSE;                                       (* STEP: 101 To PASTO -> Product Recovery End*)
                               VAR_DOS_SEQ.ITC.PROD_WaterRequestAfterProd := TRUE;                                     (* STEP: 101 To PASTO -> Water Request For Filler Rinse Afetr Production*)
```
